Yaskawa INFORM job: shotblast_perforated_cylinder_program.JBI

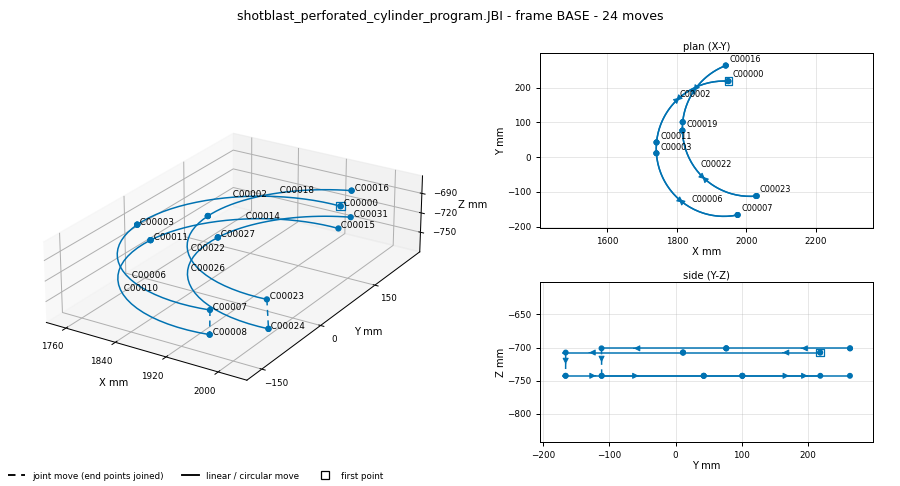
[picture p0: tool path of shotblast_perforated_cylinder_program.JBI in frame BASE, 24 of 37 moves have a stored position in this frame; points joined in program order, loops and branches not executed]
/JOB
//NAME shotblast_perforated_cylinder_program
//POS
///NPOS 32,0,32,0,0,0
///TOOL 0
///POSTYPE BASE
///RECTAN
///RCONF 0,0,0,0,0,0,0,0,0,0,0,0,0,0,0,0,0,0,0,0,0,0,0,0
C00000=1948.374666,218.096799,-707.531960,175.000000,-60.000000,-93.891690
C00001=1948.374666,218.096799,-707.531960,175.000000,-60.000000,-93.891690
C00002=1797.991079,161.841392,-707.531960,175.000000,-60.000000,-45.088731
C00003=1741.304748,11.110827,-707.531960,175.000000,-60.000000,5.000000
C00004=1741.304748,11.110827,-707.531960,175.000000,-60.000000,5.000000
C00005=1741.304748,11.110827,-707.531960,175.000000,-60.000000,5.000000
C00006=1831.955029,-140.415329,-707.531960,175.000000,-60.000000,57.911355
C00007=1975.058438,-165.968063,-707.531960,175.000000,-60.000000,101.840424
C00008=1974.459674,-166.092609,-742.628960,-175.000000,-60.000000,101.660101
C00009=1974.459674,-166.092609,-742.628960,-175.000000,-60.000000,101.660101
C00010=1801.664137,-116.965694,-742.628960,-175.000000,-60.000000,46.598295
C00011=1741.711923,42.375978,-742.628960,-175.000000,-60.000000,-5.360733
C00012=1741.711923,42.375978,-742.628960,-175.000000,-60.000000,-5.360733
C00013=1741.711923,42.375978,-742.628960,-175.000000,-60.000000,-5.360733
C00014=1812.489204,174.910453,-742.628960,-175.000000,-60.000000,-50.846306
C00015=1945.472100,218.272446,-742.628960,175.000000,-60.000000,-93.034304
C00016=1940.747537,263.152443,-701.201460,175.000000,-60.000000,-69.032105
C00017=1940.747537,263.152443,-701.201460,175.000000,-60.000000,-69.032105
C00018=1855.006292,198.530501,-701.201460,-175.000000,-60.000000,-36.958280
C00019=1816.035621,76.329608,-701.201460,-175.000000,-60.000000,5.000000
C00020=1816.035621,76.329608,-701.201460,-175.000000,-60.000000,5.000000
C00021=1816.035621,76.329608,-701.201460,-175.000000,-60.000000,5.000000
C00022=1857.341581,-38.178214,-701.201460,175.000000,-60.000000,38.088765
C00023=2027.094303,-111.898891,-701.201460,175.000000,-60.000000,94.962287
C00024=2029.628106,-111.662166,-742.654460,-175.000000,-60.000000,95.712629
C00025=2029.628106,-111.662166,-742.654460,-175.000000,-60.000000,95.712629
C00026=1843.266245,-17.633082,-742.654460,175.000000,-60.000000,30.740813
C00027=1816.886489,100.634395,-742.654460,175.000000,-60.000000,-5.592641
C00028=1816.886489,100.634395,-742.654460,175.000000,-60.000000,-5.592641
C00029=1816.886489,100.634395,-742.654460,175.000000,-60.000000,-5.592641
C00030=1843.320801,181.117867,-742.654460,-175.000000,-60.000000,-30.772268
C00031=1940.356712,263.002188,-742.654460,175.000000,-60.000000,-68.908648
///POSTYPE PULSE
///PULSE
EX00000=96256.0
EX00001=289792.0
///POSTYPE PULSE
///PULSE
EC00000=96256.0
EC00001=96256.0
EC00002=96256.0
EC00003=96256.0
EC00004=96256.0
EC00005=96256.0
EC00006=96256.0
EC00007=96256.0
EC00008=96256.0
EC00009=96256.0
EC00010=96256.0
EC00011=96256.0
EC00012=96256.0
EC00013=96256.0
EC00014=96256.0
EC00015=96256.0
EC00016=289792.0
EC00017=289792.0
EC00018=289792.0
EC00019=289792.0
EC00020=289792.0
EC00021=289792.0
EC00022=289792.0
EC00023=289792.0
EC00024=289792.0
EC00025=289792.0
EC00026=289792.0
EC00027=289792.0
EC00028=289792.0
EC00029=289792.0
EC00030=289792.0
EC00031=289792.0
//INST
///DATE 2023/08/16 12:14
///ATTR SC,RW,RJ
////FRAME BASE
///GROUP1 RB1,ST1
NOP
MOVJ P009 EX000 VJ=15.00
MOVJ C00000 EC00000 VJ=15.0
CALL JOB:SPYON
MOVC C00001 EC00001 V=150.0
MOVC C00002 EC00002 V=150.0
MOVC C00003 EC00003 V=150.0
MOVJ C00004 EC00004 VJ=15.0
MOVC C00005 EC00005 V=150.0
MOVC C00006 EC00006 V=150.0
MOVC C00007 EC00007 V=150.0
MOVJ C00008 EC00008 VJ=15.0
MOVC C00009 EC00009 V=150.0
MOVC C00010 EC00010 V=150.0
MOVC C00011 EC00011 V=150.0
MOVJ C00012 EC00012 VJ=15.0
MOVC C00013 EC00013 V=150.0
MOVC C00014 EC00014 V=150.0
MOVC C00015 EC00015 V=150.0
CALL JOB:SPYOF
MOVJ P009 VJ=15.00
MOVL P009 EX00000 V=150.0
MOVJ C00016 EC00016 VJ=15.0
CALL JOB:SPYON
MOVC C00017 EC00017 V=150.0
MOVC C00018 EC00018 V=150.0
MOVC C00019 EC00019 V=150.0
MOVJ C00020 EC00020 VJ=15.0
MOVC C00021 EC00021 V=150.0
MOVC C00022 EC00022 V=150.0
MOVC C00023 EC00023 V=150.0
MOVJ C00024 EC00024 VJ=15.0
MOVC C00025 EC00025 V=150.0
MOVC C00026 EC00026 V=150.0
MOVC C00027 EC00027 V=150.0
MOVJ C00028 EC00028 VJ=15.0
MOVC C00029 EC00029 V=150.0
MOVC C00030 EC00030 V=150.0
MOVC C00031 EC00031 V=150.0
CALL JOB:SPYOF
MOVJ P009 VJ=15.00
MOVL P009 EX00001 V=150.0
END
